{attribute 'GeneratedUsingTerminal: EL3314-0000-0018'}
{attribute addProperty BoxType "EL3314-0000-0018"}
{attribute addProperty Id "EtcSlaveTerminalBaseTC_Inputs_Channel_1AT %I*TC_Inputs_Channel_4A3944819TC_Inputs_Channel_2AT %I*TC_Inputs_Channel_4A3944819TC_Inputs_Channel_3AT %I*TC_Inputs_Channel_4A3944819TC_Inputs_Channel_4AT %I*TC_Inputs_Channel_4A3944819WcStateAT %I*WcState_9091E0EB2InfoDataAT %I*InfoData_32EB74EA10"}
{attribute addProperty CRC "1811037525"}
{attribute addProperty Size "48"}
TYPE EL3314_6BF23D55 EXTENDS EtcSlaveTerminalBase :
STRUCT
	{attribute addProperty Name "TC_Inputs_Channel_1"}
	TC_Inputs_Channel_1 : TC_Inputs_Channel_4A394481;
	{attribute addProperty Name "TC_Inputs_Channel_2"}
	TC_Inputs_Channel_2 : TC_Inputs_Channel_4A394481;
	{attribute addProperty Name "TC_Inputs_Channel_3"}
	TC_Inputs_Channel_3 : TC_Inputs_Channel_4A394481;
	{attribute addProperty Name "TC_Inputs_Channel_4"}
	TC_Inputs_Channel_4 : TC_Inputs_Channel_4A394481;
	{attribute addProperty Name "WcState"}
	WcState : WcState_9091E0EB;
	{attribute addProperty Name "InfoData"}
	InfoData : InfoData_32EB74EA;
END_STRUCT
END_TYPE

(* stored: Version 1.2.0.0, ProductVersion 3.1.4024.9
   DUT EL3314_6BF23D55: Id {66736502-2e42-42cd-adde-decbf15435ad} *)
